(* PLC project Unnamed, Unknown Unnamed 1 *)
(* stored: creationDateTime 2023-12-01T09:36:18, modificationDateTime 2023-12-01T11:01:12 *)

PROGRAM program2
  VAR
    START_BUTTON AT %QX0.0 : BOOL := 0;
    LEVEL_SENSOR AT %QX0.1 : BOOL := 0;
    CONTACT_SENSOR AT %QX0.2 : BOOL := 0;
    MOTOR AT %QX0.3 : BOOL := 0;
    NOZZLE AT %QX0.4 : BOOL := 0;
    RUN AT %QX0.5 : BOOL := 0;
  END_VAR

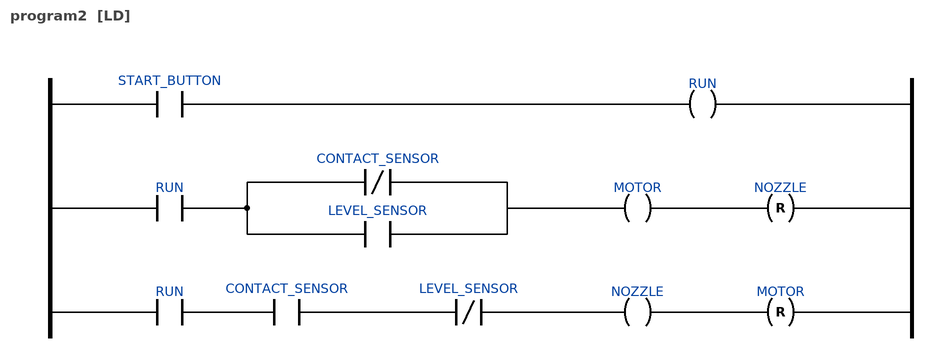
(* LD diagram, written out as Structured Text *)
RUN := START_BUTTON;
MOTOR := RUN AND (NOT CONTACT_SENSOR OR LEVEL_SENSOR);
IF RUN AND (NOT CONTACT_SENSOR OR LEVEL_SENSOR) THEN NOZZLE := FALSE; END_IF;
NOZZLE := RUN AND CONTACT_SENSOR AND NOT LEVEL_SENSOR;
IF RUN AND CONTACT_SENSOR AND NOT LEVEL_SENSOR THEN MOTOR := FALSE; END_IF;
END_PROGRAM

CONFIGURATION Config0
  RESOURCE Res0 ON PLC
    TASK task0(INTERVAL := T#20ms, PRIORITY := 0);
    PROGRAM instance0 WITH task0 : program2;
  END_RESOURCE
END_CONFIGURATION
